// TIA Portal V14 SP1 export
// export: Created 2019-04-23T05:55:44.6867831Z, ExportSetting WithDefaults, WithReadOnly, DisplayName Totally Integrated Automation Portal, DisplayVersion V14 SP1 Update 6, DisplayName TIA Portal Openness, DisplayVersion V14 SP1 Update 6, DisplayName STEP 7 Professional, DisplayVersion V14 SP1 Update 6, DisplayName WinCC Professional, DisplayVersion V14 SP1 Update 6
FUNCTION_BLOCK "D1_Divertor"   // FB1012, LAD
TITLE = Управление дивертором силосов муки
{ S7_Optimized_Access := 'FALSE' }
VERSION : 0.1
// stored: AutoNumber false, CodeModifiedDate 2019-03-26T07:08:50.0963928Z, CompileDate 2019-03-26T07:08:50.1090881Z, CreationDate 2019-02-04T08:31:08.0295361Z, InterfaceModifiedDate 2018-11-22T11:23:48.1024675Z, IsConsistent true, IsIECCheckEnabled false, IsKnowHowProtected false, ISMultiInstanceCapable true, IsWriteProtected false, LibraryConformanceStatus Warning: The object contains access to global data blocks. Warning: The block contains direct access to inputs, outputs, bit memories, indirect access to the registry or indirect access to external memory areas that are unknown at the time of compilation., ModifiedDate 2019-03-26T07:08:50.0963928Z, ParameterModified 2018-05-08T08:05:31.4379323Z, StructureModified 2018-11-22T11:23:19.1767443Z, UDAEnableTagReadback false
   VAR DB_SPECIFIC
      HMI : Struct
         CMD : Struct
            Move_Pos_1 : Bool;   // Команда переключения в позицию 1
            Spare_2 : Bool;
            Move_Pos_2 : Bool;   // Команда переключения в позицию 2
            Spare_3 : Bool;
            Spare_4 : Bool;
            Spare_5 : Bool;
            Manual : Bool;
            Reset_Error : Bool;   // Сброс ошибок
         END_STRUCT;
         DATA : Struct
            StatusWord : Word;   // Статус состояния
            Pos1_Time : DInt := 5;   // Время контроля срабатывания датчика 1 / Время контроля срабатывания датчика 1 (сек)
            Pos2_Time : DInt := 5;   // Время контроля срабатывания датчика 2 / Время контроля срабатывания датчика 2 (сек)
         END_STRUCT;
      END_STRUCT;
   END_VAR
   VAR
      Two_Valve : "Two_Valve_Manag";
   END_VAR
   VAR DB_SPECIFIC
      ResetErr : Bool;   // сброс ошибок
      General_cond_OK : Bool;   // Разрешение работы
      ManCmd_Silos_1 : Bool;   // Команда ручного переключения дивертора на силос 1
      ManCmd_Silos_2 : Bool;   // Команда ручного переключения дивертора на силос 2
      AutoCmd_Silos_1 : Bool;   // Команда автом. переключения дивертора на силос 1
      AutoCmd_Silos_2 : Bool;   // Команда автом. переключения дивертора на силос 2
      Pos1_Time : Time;   // Время контроля перемещения в позицию 1
      Pos2_Time : Time;   // Время контроля перемещения в позицию 2
   END_VAR
   VAR_TEMP   // added for the SCL form of the ladder/FBD networks
      _w1 : Bool;
   END_VAR
BEGIN

REGION Network 1: Сброс ошибок
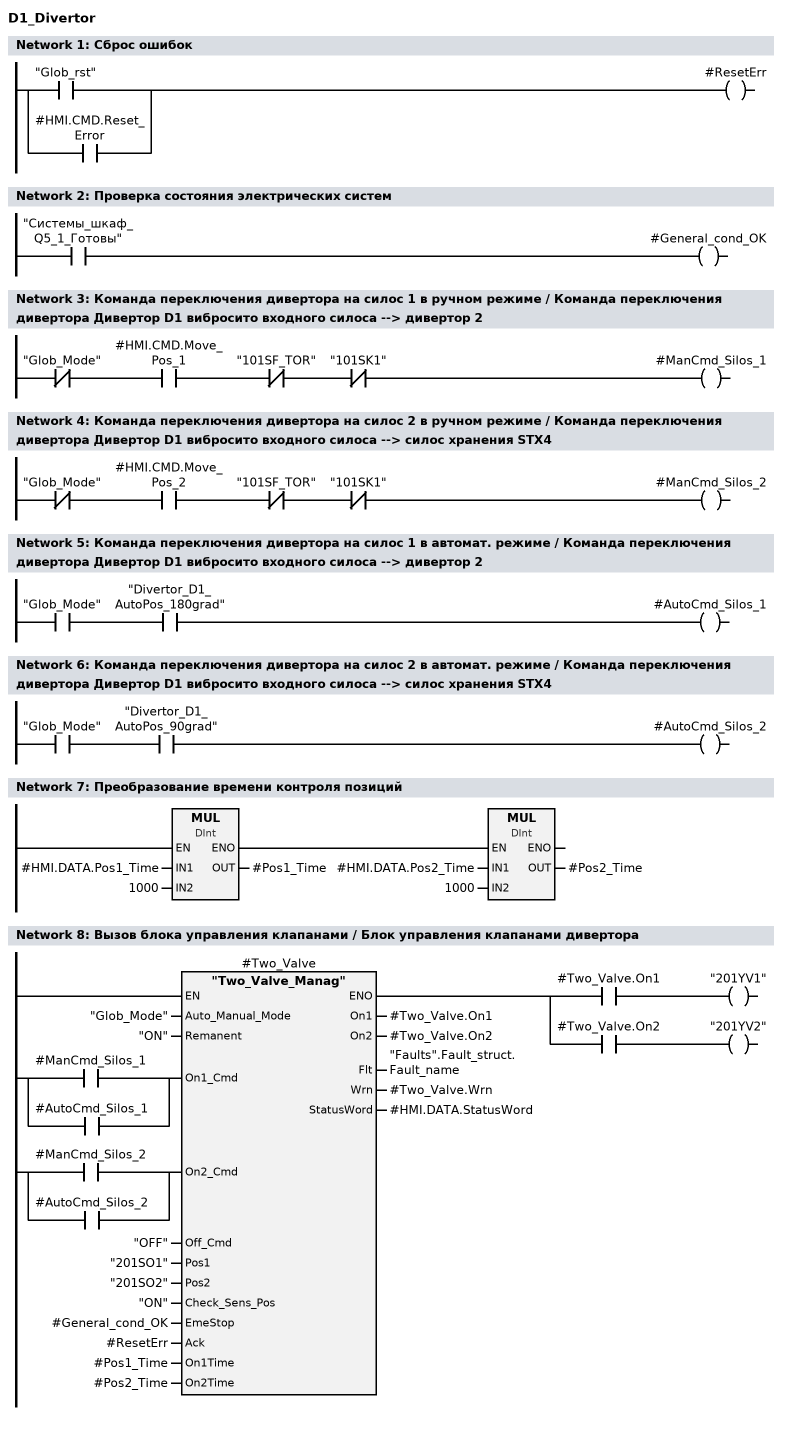
   RUNG wire#powerrail
      Contact( "Glob_rst" )
      wire#w1
      Coil( #ResetErr )
   END_RUNG
   RUNG wire#powerrail
      Contact( #HMI.CMD.Reset_Error )
   END_RUNG wire#w1
   // the same network as SCL:
   #ResetErr := "Glob_rst" OR #HMI.CMD.Reset_Error;
END_REGION

REGION Network 2: Проверка состояния электрических систем
   RUNG wire#powerrail
      Contact( "Системы_шкаф_Q5_1_Готовы" )
      Coil( #General_cond_OK )
   END_RUNG
   // the same network as SCL:
   #General_cond_OK := "Системы_шкаф_Q5_1_Готовы";
END_REGION

REGION Network 3: Команда переключения дивертора на силос 1 в ручном режиме / Команда переключения дивертора Дивертор D1 вибросито входного силоса --> дивертор 2
   RUNG wire#powerrail
      I_Contact( "Glob_Mode" )
      Contact( #HMI.CMD.Move_Pos_1 )
      I_Contact( "101SF_TOR" )
      I_Contact( "101SK1" )
      Coil( #ManCmd_Silos_1 )
   END_RUNG
   // the same network as SCL:
   #ManCmd_Silos_1 := NOT "Glob_Mode" AND #HMI.CMD.Move_Pos_1 AND NOT "101SF_TOR" AND NOT "101SK1";
END_REGION

REGION Network 4: Команда переключения дивертора на силос 2 в ручном режиме / Команда переключения дивертора Дивертор D1 вибросито входного силоса --> силос хранения STX4
   RUNG wire#powerrail
      I_Contact( "Glob_Mode" )
      Contact( #HMI.CMD.Move_Pos_2 )
      I_Contact( "101SF_TOR" )
      I_Contact( "101SK1" )
      Coil( #ManCmd_Silos_2 )
   END_RUNG
   // the same network as SCL:
   #ManCmd_Silos_2 := NOT "Glob_Mode" AND #HMI.CMD.Move_Pos_2 AND NOT "101SF_TOR" AND NOT "101SK1";
END_REGION

REGION Network 5: Команда переключения дивертора на силос 1 в автомат. режиме / Команда переключения дивертора Дивертор D1 вибросито входного силоса --> дивертор 2
   RUNG wire#powerrail
      Contact( "Glob_Mode" )
      Contact( "Divertor_D1_AutoPos_180grad" )
      Coil( #AutoCmd_Silos_1 )
   END_RUNG
   // the same network as SCL:
   #AutoCmd_Silos_1 := "Glob_Mode" AND "Divertor_D1_AutoPos_180grad";
END_REGION

REGION Network 6: Команда переключения дивертора на силос 2 в автомат. режиме / Команда переключения дивертора Дивертор D1 вибросито входного силоса --> силос хранения STX4
   RUNG wire#powerrail
      Contact( "Glob_Mode" )
      Contact( "Divertor_D1_AutoPos_90grad" )
      Coil( #AutoCmd_Silos_2 )
   END_RUNG
   // the same network as SCL:
   #AutoCmd_Silos_2 := "Glob_Mode" AND "Divertor_D1_AutoPos_90grad";
END_REGION

REGION Network 7: Преобразование времени контроля позиций
   RUNG wire#powerrail
      { S7_Templates := "SrcType := DInt"; S7_GenerateENO := "TRUE" } Mul(in1 := #HMI.DATA.Pos1_Time, in2 := 1000, out => #Pos1_Time)
      { S7_Templates := "SrcType := DInt"; S7_GenerateENO := "TRUE" } Mul(in1 := #HMI.DATA.Pos2_Time, in2 := 1000, out => #Pos2_Time)
   END_RUNG
   // the same network as SCL:
   // ENO of a box is taken as its EN; it also drops when the box reports an error
   #Pos1_Time := #HMI.DATA.Pos1_Time * 1000;
   #Pos2_Time := #HMI.DATA.Pos2_Time * 1000;
END_REGION

REGION Network 8: Вызов блока управления клапанами / Блок управления клапанами дивертора
   RUNG wire#powerrail
      #Two_Valve(On1_Cmd := wire#w1, On2_Cmd := wire#w2, Auto_Manual_Mode := "Glob_Mode", Remanent := "ON", Off_Cmd := "OFF", Pos1 := "201SO1", Pos2 := "201SO2", Check_Sens_Pos := "ON", EmeStop := #General_cond_OK, Ack := #ResetErr, On1Time := #Pos1_Time, On2Time := #Pos2_Time, On1 => #Two_Valve.On1, On2 => #Two_Valve.On2, Flt => "Faults".Fault_struct.Fault_name, Wrn => #Two_Valve.Wrn, StatusWord => #HMI.DATA.StatusWord)
      wire#w3
      Contact( #Two_Valve.On1 )
      Coil( "201YV1" )
   END_RUNG
   RUNG wire#powerrail
      Contact( #ManCmd_Silos_1 )
   END_RUNG wire#w1
   RUNG wire#powerrail
      Contact( #AutoCmd_Silos_1 )
   END_RUNG wire#w1
   RUNG wire#powerrail
      Contact( #ManCmd_Silos_2 )
   END_RUNG wire#w2
   RUNG wire#powerrail
      Contact( #AutoCmd_Silos_2 )
   END_RUNG wire#w2
   RUNG wire#w3
      Contact( #Two_Valve.On2 )
      Coil( "201YV2" )
   END_RUNG
   // the same network as SCL:
   #Two_Valve(Auto_Manual_Mode := "Glob_Mode",   // "Two_Valve_Manag"
              Remanent := "ON",
              On1_Cmd := #ManCmd_Silos_1 OR #AutoCmd_Silos_1,
              On2_Cmd := #ManCmd_Silos_2 OR #AutoCmd_Silos_2,
              Off_Cmd := "OFF",
              Pos1 := "201SO1",
              Pos2 := "201SO2",
              Check_Sens_Pos := "ON",
              EmeStop := #General_cond_OK,
              Ack := #ResetErr,
              On1Time := #Pos1_Time,
              On2Time := #Pos2_Time,
              On1 => #Two_Valve.On1,
              On2 => #Two_Valve.On2,
              Flt => "Faults".Fault_struct.Fault_name,
              Wrn => #Two_Valve.Wrn,
              StatusWord => #HMI.DATA.StatusWord,
              ENO => #_w1);
   "201YV1" := #_w1 AND #Two_Valve.On1;
   "201YV2" := #_w1 AND #Two_Valve.On2;
END_REGION
END_FUNCTION_BLOCK
